KUKA KRL data list: Class_EAxisAsync.dat

&ACCESS RV1
&REL 4
&PARAM DISKPATH = KRC:\R1\FUNCTION
DEFDAT Class_EAxisAsync PUBLIC
REAL lastEAxis[6] ; Gun motor positon on decouple
lastEAxis[1]=33.2811279
lastEAxis[2]=18.3915939
lastEAxis[3]=18.7621956
lastEAxis[4]=20.0000
lastEAxis[5]=0.0
lastEAxis[6]=0.0
ENDDAT
